(* LS Electric XG5000 project: CLRCAP *)
(* PLC LSPLC *)

PROGRAM NewProgram (* task: 스캔 프로그램 *)
VAR
    _t1 : DINT;
    _t2 : DINT;
    _t3 : DINT;
    _t4 : BOOL;
END_VAR

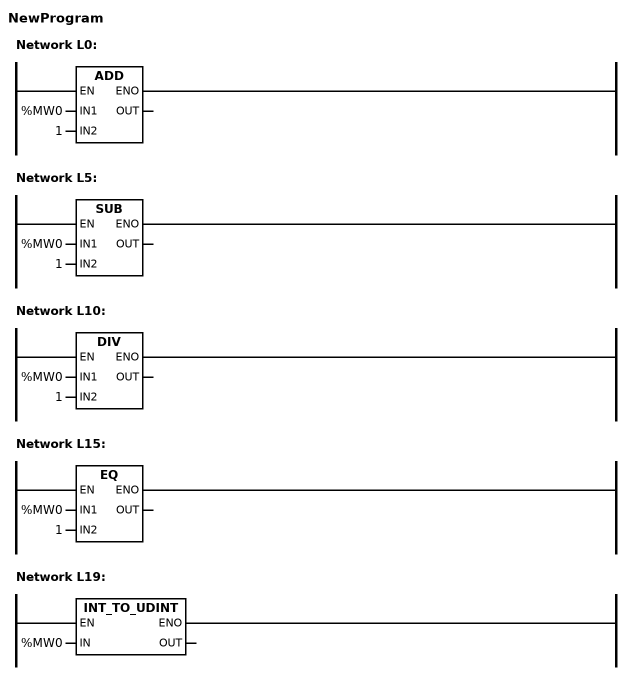
(* Rung L0 *)
_t1 := %MW0 + 1;
(* Rung L5 *)
_t2 := %MW0 - 1;
(* Rung L10 *)
_t3 := %MW0 / 1;
(* Rung L15 *)
_t4 := %MW0 = 1;
(* Rung L19 *)
INT_TO_UDINT(%MW0);
END_PROGRAM